(* Logix 5000 project; controller Amvex_Thorpe_Flowmeter vendor 1 type 14 code 106 rev 33.13; software revision 33.01; part 16 of 16 *)
(* tags used below, declared in another part *)
   Auto_Seq : SEQ;
   FAULTED : DINT;
   MODE : MODE;
   ID0_InputDataLength : MESSAGE;   // Message Command Input Data Data Length
   ID0_LengthParameterdata : MESSAGE;   // Message Command Parameter Data Length
   ID0_MSG_Diagnostic : MESSAGE;   // Message Get Diagnosis Module
   ID0_MSG_ProcessAlarm : MESSAGE;   // Message Get Get Process Alram Module
   ID0_OutputDataLength : MESSAGE;   // Message Command Output Data Data Length
   ID0_ReceiveMSG1 : MESSAGE;   // Message Command Parameter Receive Data
   ID0_ReceiveMSG2 : MESSAGE;   // Message Command Parameter Receive Data
   ID0_ReceiveMSG3 : MESSAGE;   // Message Command Parameter Receive Data
   ID0_SendMSG1 : MESSAGE;   // Message Command Parameter Send Data
   ID0_SendMSG2 : MESSAGE;   // Message Command Parameter Send Data
   ID0_SendMSG3 : MESSAGE;   // Message Command Parameter Send Data
   In_Cycle : BOOL;
   RCP1 : RCP1;
   RCP1_00 : UDT_ID0;
(* RPC1_Main, continued *)

ROUTINE R07_MODE   (* ladder *)
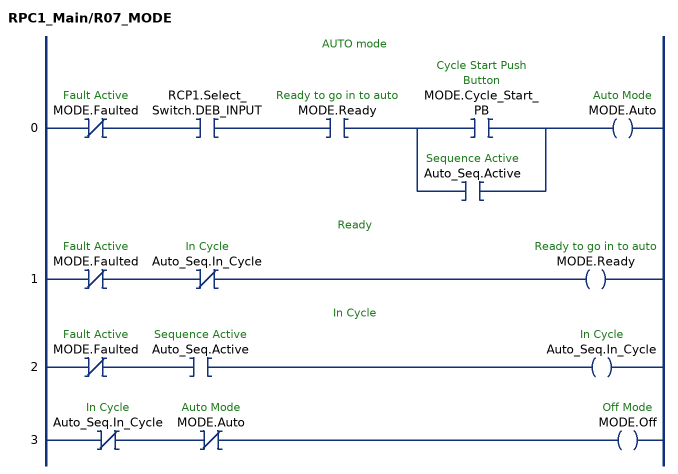
   // AUTO mode
   0: XIO(MODE.Faulted)XIC(RCP1.Select_Switch.DEB_INPUT)XIC(MODE.Ready)[XIC(MODE.Cycle_Start_PB) ,XIC(Auto_Seq.Active) ]OTE(MODE.Auto);
   // Ready
   1: XIO(MODE.Faulted)XIO(Auto_Seq.In_Cycle)OTE(MODE.Ready);
   // In Cycle
   2: XIO(MODE.Faulted)XIC(Auto_Seq.Active)OTE(Auto_Seq.In_Cycle);
   3: XIO(Auto_Seq.In_Cycle)XIO(MODE.Auto)OTE(MODE.Off);
END_ROUTINE

ROUTINE RCP1_00_RACK_IO   (* ladder *)
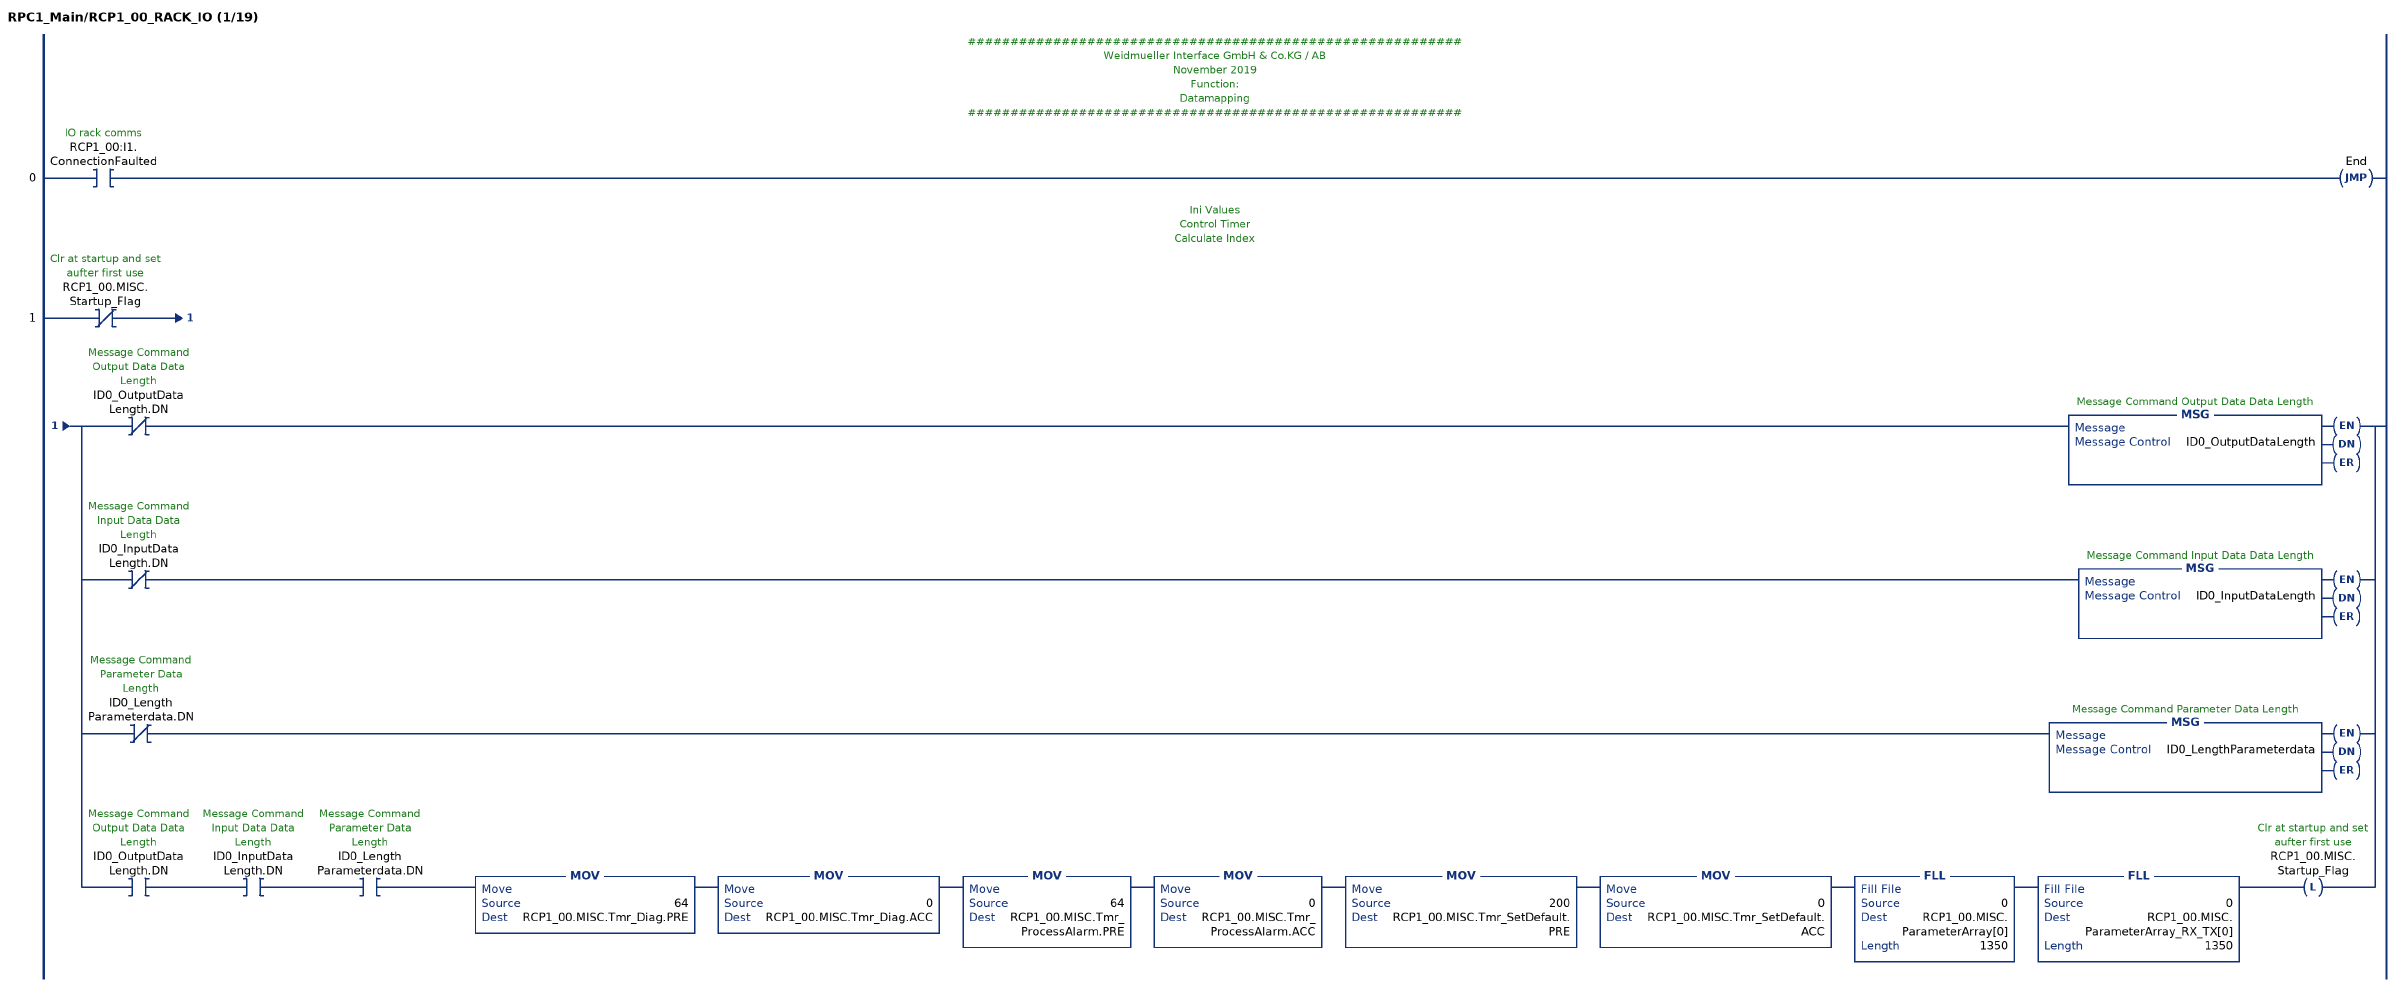
   // ##########################################################
   // Weidmueller Interface GmbH & Co.KG / AB
   // November 2019
   // Function:
   // Datamapping
   // ##########################################################
   0: XIC(RCP1_00:I1.ConnectionFaulted)JMP(End);
   // Ini Values
   // Control Timer
   // Calculate Index
   1: XIO(RCP1_00.MISC.Startup_Flag)[[XIO(ID0_OutputDataLength.DN) MSG(ID0_OutputDataLength) ,XIO(ID0_InputDataLength.DN) MSG(ID0_InputDataLength) ,XIO(ID0_LengthParameterdata.DN) MSG(ID0_LengthParameterdata) ] ,XIC(ID0_OutputDataLength.DN) XIC(ID0_InputDataLength.DN) XIC(ID0_LengthParameterdata.DN) MOV(64,RCP1_00.MISC.Tmr_Diag.PRE) MOV(0,RCP1_00.MISC.Tmr_Diag.ACC) MOV(64,RCP1_00.MISC.Tmr_ProcessAlarm.PRE) MOV(0,RCP1_00.MISC.Tmr_ProcessAlarm.ACC) MOV(200,RCP1_00.MISC.Tmr_SetDefault.PRE) MOV(0,RCP1_00.MISC.Tmr_SetDefault.ACC) FLL(0,RCP1_00.MISC.ParameterArray[0],1350) FLL(0,RCP1_00.MISC.ParameterArray_RX_TX[0],1350) OTL(RCP1_00.MISC.Startup_Flag) ];
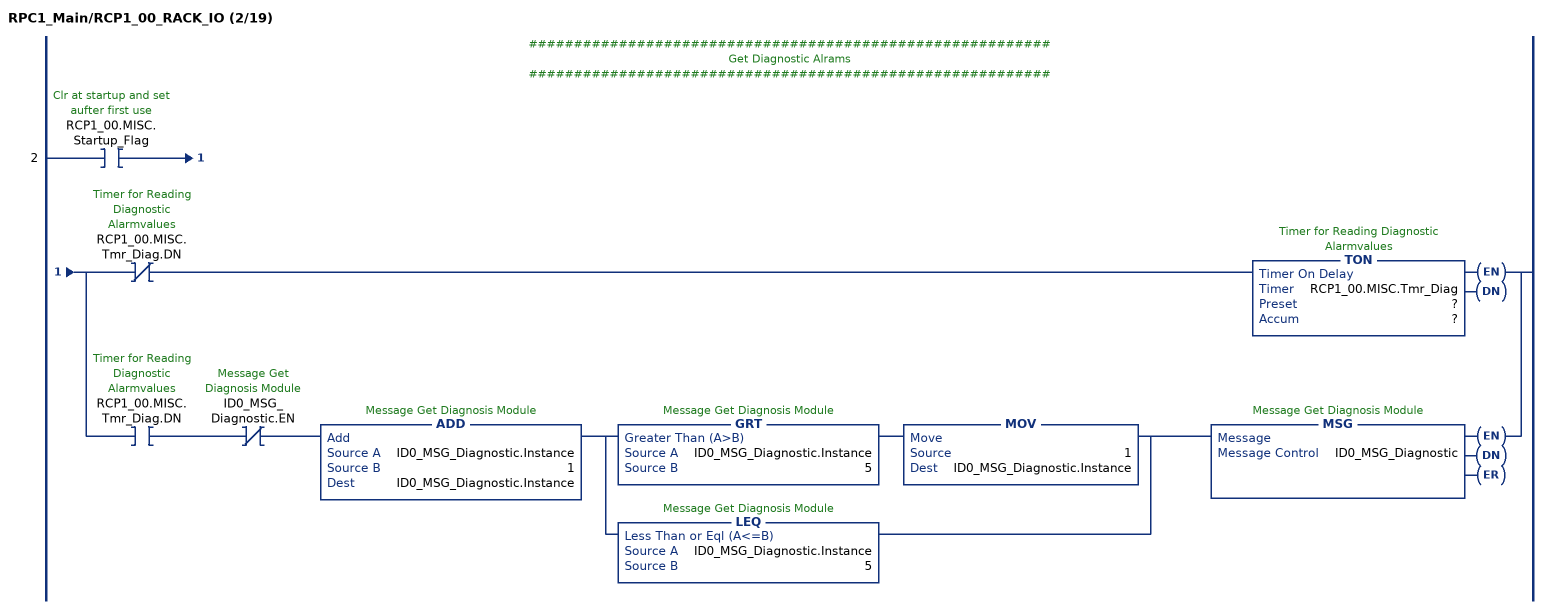
   // ##########################################################
   // Get Diagnostic Alrams
   // ##########################################################
   2: XIC(RCP1_00.MISC.Startup_Flag)[XIO(RCP1_00.MISC.Tmr_Diag.DN) TON(RCP1_00.MISC.Tmr_Diag,?,?) ,XIC(RCP1_00.MISC.Tmr_Diag.DN) XIO(ID0_MSG_Diagnostic.EN) ADD(ID0_MSG_Diagnostic.Instance,1,ID0_MSG_Diagnostic.Instance) [GRT(ID0_MSG_Diagnostic.Instance,5) MOV(1,ID0_MSG_Diagnostic.Instance) ,LEQ(ID0_MSG_Diagnostic.Instance,5) ] MSG(ID0_MSG_Diagnostic) ];
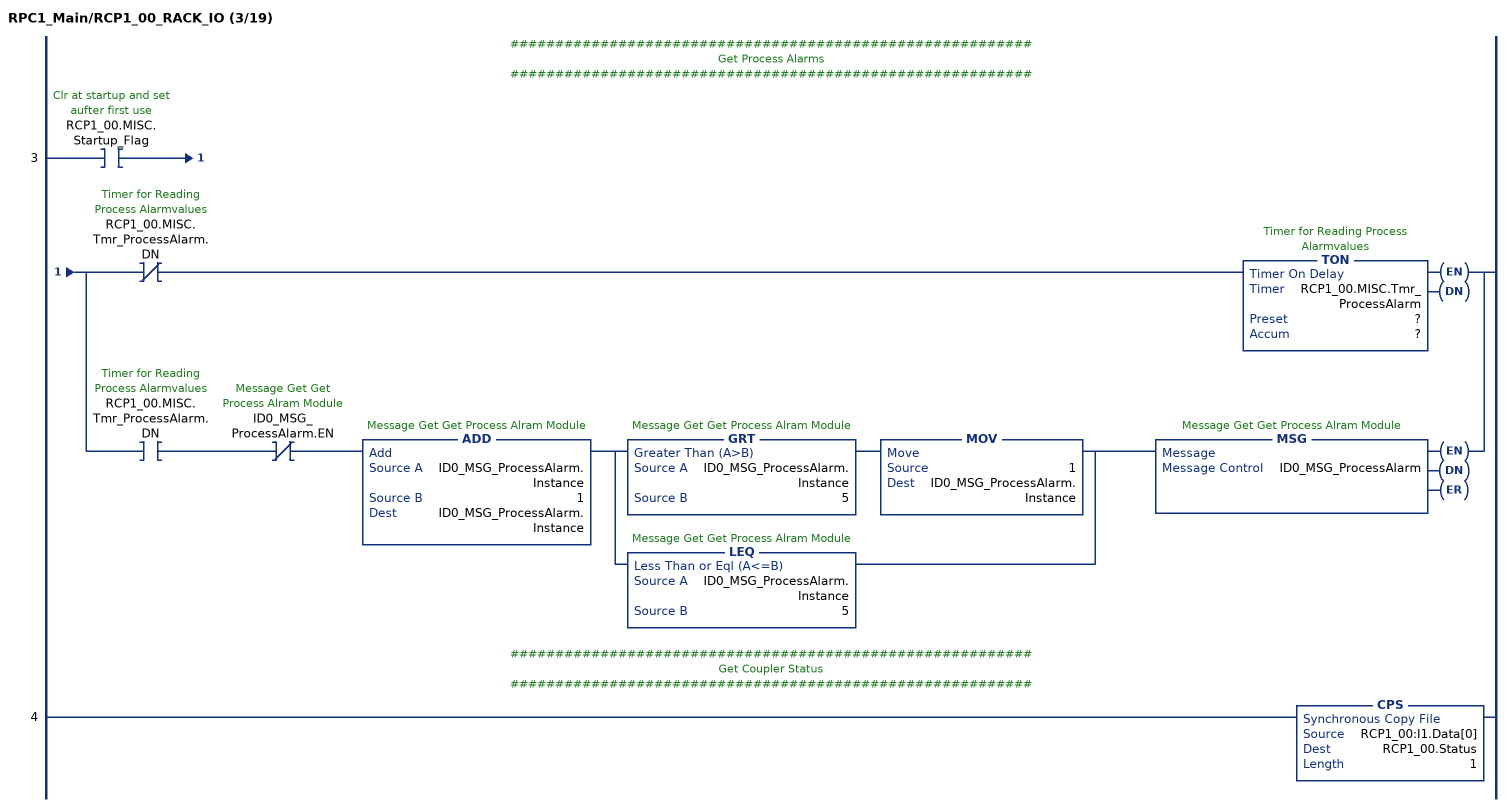
   // ##########################################################
   // Get Process Alarms
   // ##########################################################
   3: XIC(RCP1_00.MISC.Startup_Flag)[XIO(RCP1_00.MISC.Tmr_ProcessAlarm.DN) TON(RCP1_00.MISC.Tmr_ProcessAlarm,?,?) ,XIC(RCP1_00.MISC.Tmr_ProcessAlarm.DN) XIO(ID0_MSG_ProcessAlarm.EN) ADD(ID0_MSG_ProcessAlarm.Instance,1,ID0_MSG_ProcessAlarm.Instance) [GRT(ID0_MSG_ProcessAlarm.Instance,5) MOV(1,ID0_MSG_ProcessAlarm.Instance) ,LEQ(ID0_MSG_ProcessAlarm.Instance,5) ] MSG(ID0_MSG_ProcessAlarm) ];
   // ##########################################################
   // Get Coupler Status
   // ##########################################################
   4: CPS(RCP1_00:I1.Data[0],RCP1_00.Status,1);
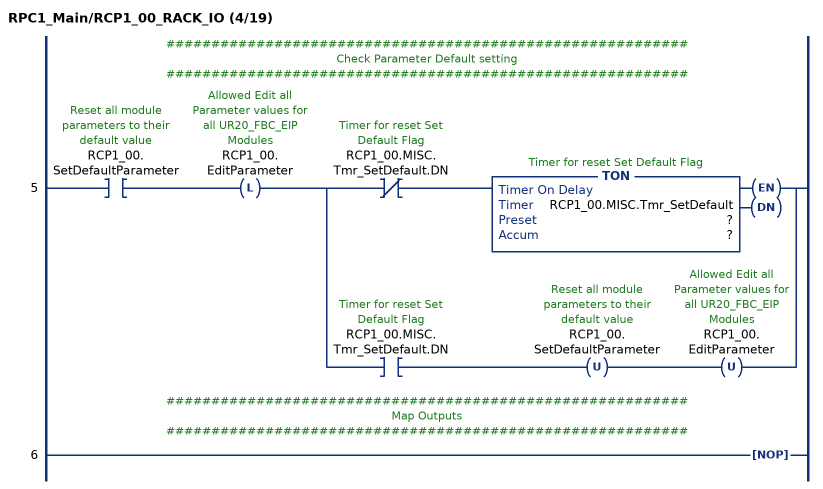
   // ##########################################################
   // Check Parameter Default setting
   // ##########################################################
   5: XIC(RCP1_00.SetDefaultParameter)OTL(RCP1_00.EditParameter)[XIO(RCP1_00.MISC.Tmr_SetDefault.DN) TON(RCP1_00.MISC.Tmr_SetDefault,?,?) ,XIC(RCP1_00.MISC.Tmr_SetDefault.DN) OTU(RCP1_00.SetDefaultParameter) OTU(RCP1_00.EditParameter) ];
   // ##########################################################
   // Map Outputs
   // ##########################################################
   6: NOP();
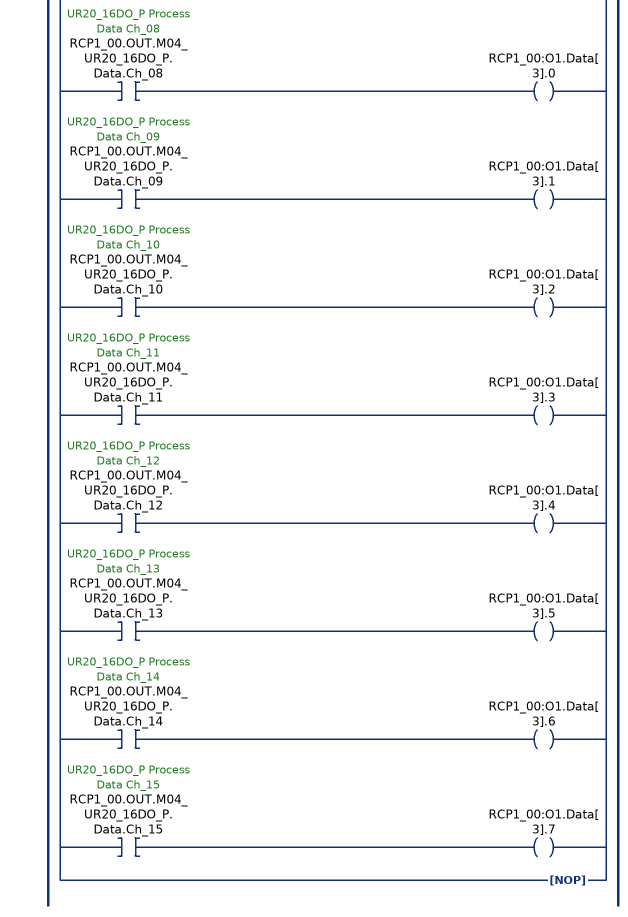
   // Map
   //  UR20_16DO_P
   //  Module No 4
   //  Process Data
   //  Outputs
   7: [NOP() ,XIC(RCP1_00.OUT.M04_UR20_16DO_P.Data.Ch_00) OTE(RCP1_00:O1.Data[2].0) ,XIC(RCP1_00.OUT.M04_UR20_16DO_P.Data.Ch_01) OTE(RCP1_00:O1.Data[2].1) ,XIC(RCP1_00.OUT.M04_UR20_16DO_P.Data.Ch_02) OTE(RCP1_00:O1.Data[2].2) ,XIC(RCP1_00.OUT.M04_UR20_16DO_P.Data.Ch_03) OTE(RCP1_00:O1.Data[2].3) ,XIC(RCP1_00.OUT.M04_UR20_16DO_P.Data.Ch_04) OTE(RCP1_00:O1.Data[2].4) ,XIC(RCP1_00.OUT.M04_UR20_16DO_P.Data.Ch_05) OTE(RCP1_00:O1.Data[2].5) ,XIC(RCP1_00.OUT.M04_UR20_16DO_P.Data.Ch_06) OTE(RCP1_00:O1.Data[2].6) ,XIC(RCP1_00.OUT.M04_UR20_16DO_P.Data.Ch_07) OTE(RCP1_00:O1.Data[2].7) ,XIC(RCP1_00.OUT.M04_UR20_16DO_P.Data.Ch_08) OTE(RCP1_00:O1.Data[3].0) ,XIC(RCP1_00.OUT.M04_UR20_16DO_P.Data.Ch_09) OTE(RCP1_00:O1.Data[3].1) ,XIC(RCP1_00.OUT.M04_UR20_16DO_P.Data.Ch_10) OTE(RCP1_00:O1.Data[3].2) ,XIC(RCP1_00.OUT.M04_UR20_16DO_P.Data.Ch_11) OTE(RCP1_00:O1.Data[3].3) ,XIC(RCP1_00.OUT.M04_UR20_16DO_P.Data.Ch_12) OTE(RCP1_00:O1.Data[3].4) ,XIC(RCP1_00.OUT.M04_UR20_16DO_P.Data.Ch_13) OTE(RCP1_00:O1.Data[3].5) ,XIC(RCP1_00.OUT.M04_UR20_16DO_P.Data.Ch_14) OTE(RCP1_00:O1.Data[3].6) ,XIC(RCP1_00.OUT.M04_UR20_16DO_P.Data.Ch_15) OTE(RCP1_00:O1.Data[3].7) ,NOP() ];
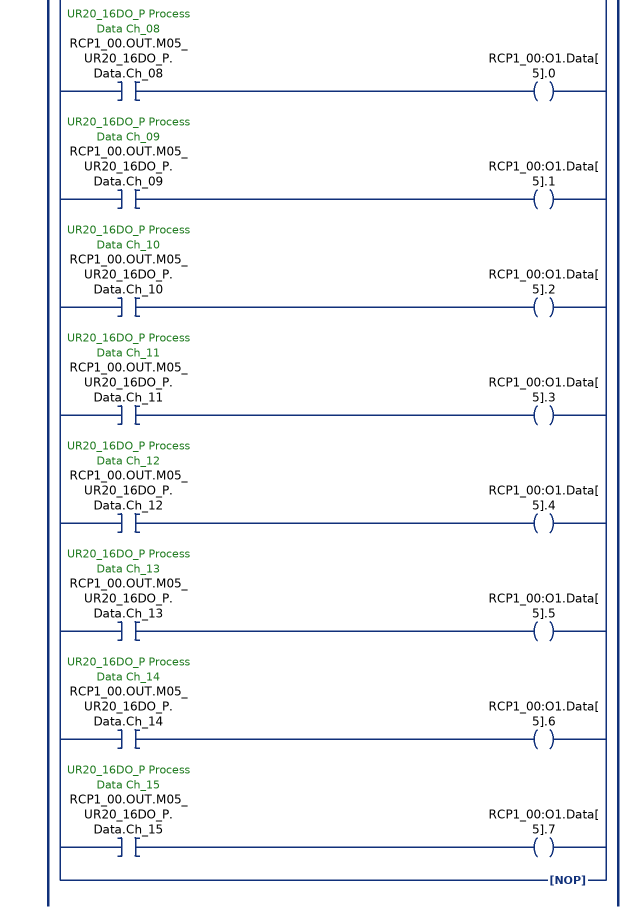
   // Map
   //  UR20_16DO_P
   //  Module No 5
   //  Process Data
   //  Outputs
   8: [NOP() ,XIC(RCP1_00.OUT.M05_UR20_16DO_P.Data.Ch_00) OTE(RCP1_00:O1.Data[4].0) ,XIC(RCP1_00.OUT.M05_UR20_16DO_P.Data.Ch_01) OTE(RCP1_00:O1.Data[4].1) ,XIC(RCP1_00.OUT.M05_UR20_16DO_P.Data.Ch_02) OTE(RCP1_00:O1.Data[4].2) ,XIC(RCP1_00.OUT.M05_UR20_16DO_P.Data.Ch_03) OTE(RCP1_00:O1.Data[4].3) ,XIC(RCP1_00.OUT.M05_UR20_16DO_P.Data.Ch_04) OTE(RCP1_00:O1.Data[4].4) ,XIC(RCP1_00.OUT.M05_UR20_16DO_P.Data.Ch_05) OTE(RCP1_00:O1.Data[4].5) ,XIC(RCP1_00.OUT.M05_UR20_16DO_P.Data.Ch_06) OTE(RCP1_00:O1.Data[4].6) ,XIC(RCP1_00.OUT.M05_UR20_16DO_P.Data.Ch_07) OTE(RCP1_00:O1.Data[4].7) ,XIC(RCP1_00.OUT.M05_UR20_16DO_P.Data.Ch_08) OTE(RCP1_00:O1.Data[5].0) ,XIC(RCP1_00.OUT.M05_UR20_16DO_P.Data.Ch_09) OTE(RCP1_00:O1.Data[5].1) ,XIC(RCP1_00.OUT.M05_UR20_16DO_P.Data.Ch_10) OTE(RCP1_00:O1.Data[5].2) ,XIC(RCP1_00.OUT.M05_UR20_16DO_P.Data.Ch_11) OTE(RCP1_00:O1.Data[5].3) ,XIC(RCP1_00.OUT.M05_UR20_16DO_P.Data.Ch_12) OTE(RCP1_00:O1.Data[5].4) ,XIC(RCP1_00.OUT.M05_UR20_16DO_P.Data.Ch_13) OTE(RCP1_00:O1.Data[5].5) ,XIC(RCP1_00.OUT.M05_UR20_16DO_P.Data.Ch_14) OTE(RCP1_00:O1.Data[5].6) ,XIC(RCP1_00.OUT.M05_UR20_16DO_P.Data.Ch_15) OTE(RCP1_00:O1.Data[5].7) ,NOP() ];
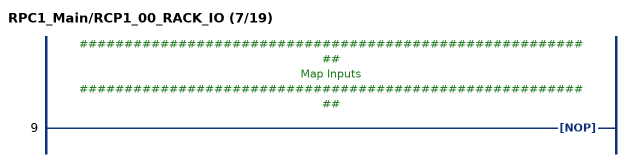
   // ##########################################################
   // Map Inputs
   // ##########################################################
   9: NOP();
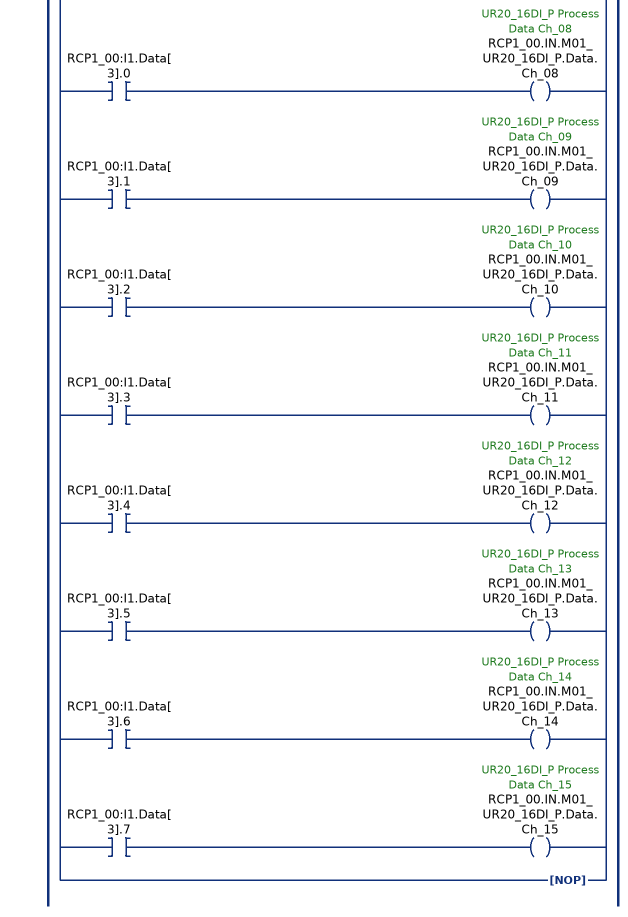
   // Map
   //  UR20_16DI_P
   //  Module No 1
   //  Process Data
   //  Inputs
   10: [NOP() ,XIC(RCP1_00:I1.Data[2].0) OTE(RCP1_00.IN.M01_UR20_16DI_P.Data.Ch_00) ,XIC(RCP1_00:I1.Data[2].1) OTE(RCP1_00.IN.M01_UR20_16DI_P.Data.Ch_01) ,XIC(RCP1_00:I1.Data[2].2) OTE(RCP1_00.IN.M01_UR20_16DI_P.Data.Ch_02) ,XIC(RCP1_00:I1.Data[2].3) OTE(RCP1_00.IN.M01_UR20_16DI_P.Data.Ch_03) ,XIC(RCP1_00:I1.Data[2].4) OTE(RCP1_00.IN.M01_UR20_16DI_P.Data.Ch_04) ,XIC(RCP1_00:I1.Data[2].5) OTE(RCP1_00.IN.M01_UR20_16DI_P.Data.Ch_05) ,XIC(RCP1_00:I1.Data[2].6) OTE(RCP1_00.IN.M01_UR20_16DI_P.Data.Ch_06) ,XIC(RCP1_00:I1.Data[2].7) OTE(RCP1_00.IN.M01_UR20_16DI_P.Data.Ch_07) ,XIC(RCP1_00:I1.Data[3].0) OTE(RCP1_00.IN.M01_UR20_16DI_P.Data.Ch_08) ,XIC(RCP1_00:I1.Data[3].1) OTE(RCP1_00.IN.M01_UR20_16DI_P.Data.Ch_09) ,XIC(RCP1_00:I1.Data[3].2) OTE(RCP1_00.IN.M01_UR20_16DI_P.Data.Ch_10) ,XIC(RCP1_00:I1.Data[3].3) OTE(RCP1_00.IN.M01_UR20_16DI_P.Data.Ch_11) ,XIC(RCP1_00:I1.Data[3].4) OTE(RCP1_00.IN.M01_UR20_16DI_P.Data.Ch_12) ,XIC(RCP1_00:I1.Data[3].5) OTE(RCP1_00.IN.M01_UR20_16DI_P.Data.Ch_13) ,XIC(RCP1_00:I1.Data[3].6) OTE(RCP1_00.IN.M01_UR20_16DI_P.Data.Ch_14) ,XIC(RCP1_00:I1.Data[3].7) OTE(RCP1_00.IN.M01_UR20_16DI_P.Data.Ch_15) ,NOP() ];
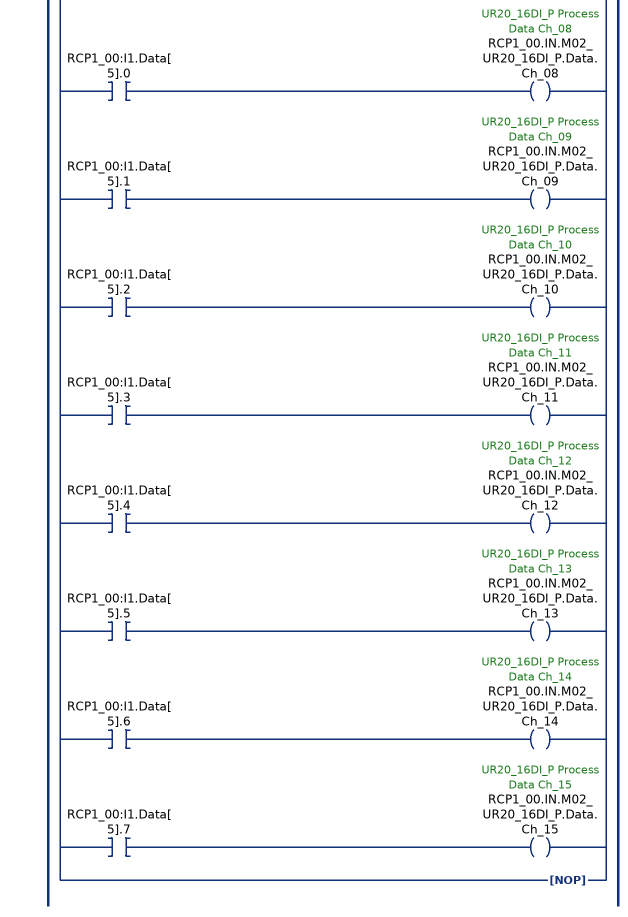
   // Map
   //  UR20_16DI_P
   //  Module No 2
   //  Process Data
   //  Inputs
   11: [NOP() ,XIC(RCP1_00:I1.Data[4].0) OTE(RCP1_00.IN.M02_UR20_16DI_P.Data.Ch_00) ,XIC(RCP1_00:I1.Data[4].1) OTE(RCP1_00.IN.M02_UR20_16DI_P.Data.Ch_01) ,XIC(RCP1_00:I1.Data[4].2) OTE(RCP1_00.IN.M02_UR20_16DI_P.Data.Ch_02) ,XIC(RCP1_00:I1.Data[4].3) OTE(RCP1_00.IN.M02_UR20_16DI_P.Data.Ch_03) ,XIC(RCP1_00:I1.Data[4].4) OTE(RCP1_00.IN.M02_UR20_16DI_P.Data.Ch_04) ,XIC(RCP1_00:I1.Data[4].5) OTE(RCP1_00.IN.M02_UR20_16DI_P.Data.Ch_05) ,XIC(RCP1_00:I1.Data[4].6) OTE(RCP1_00.IN.M02_UR20_16DI_P.Data.Ch_06) ,XIC(RCP1_00:I1.Data[4].7) OTE(RCP1_00.IN.M02_UR20_16DI_P.Data.Ch_07) ,XIC(RCP1_00:I1.Data[5].0) OTE(RCP1_00.IN.M02_UR20_16DI_P.Data.Ch_08) ,XIC(RCP1_00:I1.Data[5].1) OTE(RCP1_00.IN.M02_UR20_16DI_P.Data.Ch_09) ,XIC(RCP1_00:I1.Data[5].2) OTE(RCP1_00.IN.M02_UR20_16DI_P.Data.Ch_10) ,XIC(RCP1_00:I1.Data[5].3) OTE(RCP1_00.IN.M02_UR20_16DI_P.Data.Ch_11) ,XIC(RCP1_00:I1.Data[5].4) OTE(RCP1_00.IN.M02_UR20_16DI_P.Data.Ch_12) ,XIC(RCP1_00:I1.Data[5].5) OTE(RCP1_00.IN.M02_UR20_16DI_P.Data.Ch_13) ,XIC(RCP1_00:I1.Data[5].6) OTE(RCP1_00.IN.M02_UR20_16DI_P.Data.Ch_14) ,XIC(RCP1_00:I1.Data[5].7) OTE(RCP1_00.IN.M02_UR20_16DI_P.Data.Ch_15) ,NOP() ];
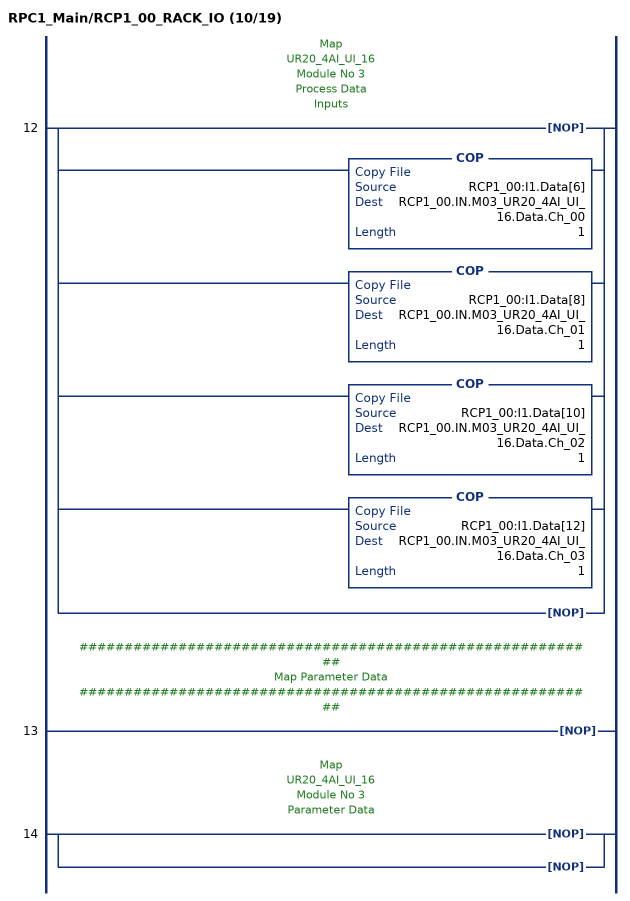
   // Map
   //  UR20_4AI_UI_16
   //  Module No 3
   //  Process Data
   //  Inputs
   12: [NOP() ,COP(RCP1_00:I1.Data[6],RCP1_00.IN.M03_UR20_4AI_UI_16.Data.Ch_00,1) ,COP(RCP1_00:I1.Data[8],RCP1_00.IN.M03_UR20_4AI_UI_16.Data.Ch_01,1) ,COP(RCP1_00:I1.Data[10],RCP1_00.IN.M03_UR20_4AI_UI_16.Data.Ch_02,1) ,COP(RCP1_00:I1.Data[12],RCP1_00.IN.M03_UR20_4AI_UI_16.Data.Ch_03,1) ,NOP() ];
   // ##########################################################
   // Map Parameter Data
   // ##########################################################
   13: NOP();
   // Map
   //  UR20_4AI_UI_16
   //  Module No 3
   //  Parameter Data
   14: [NOP() ,NOP() ];
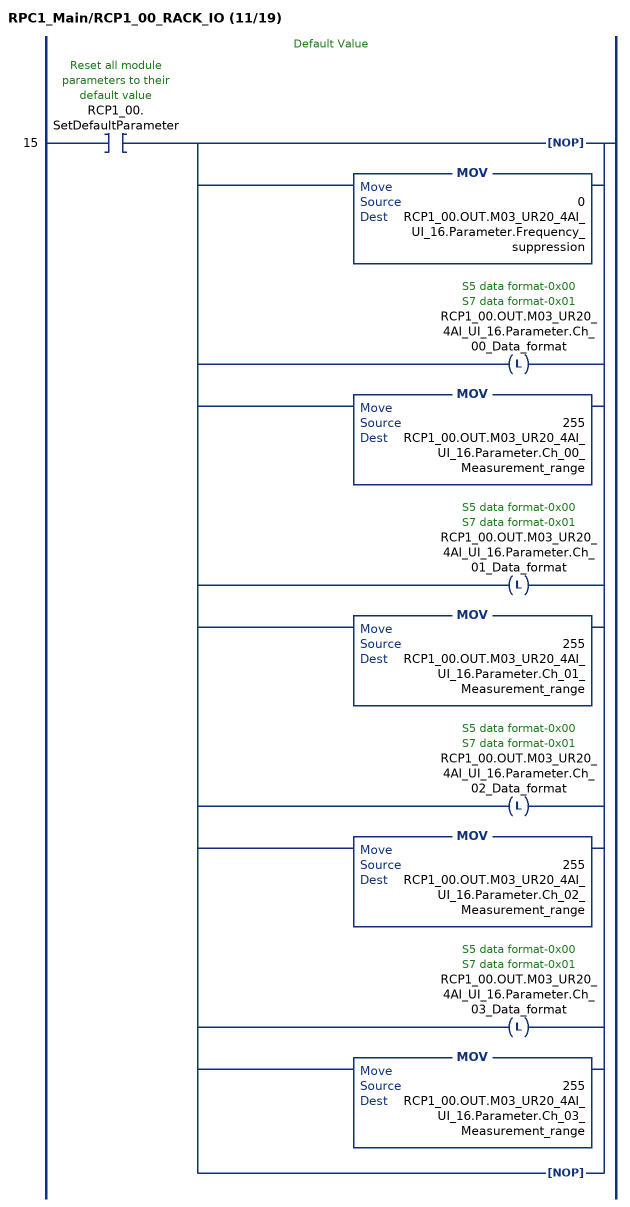
   // Default Value
   15: XIC(RCP1_00.SetDefaultParameter)[NOP() ,MOV(0,RCP1_00.OUT.M03_UR20_4AI_UI_16.Parameter.Frequency_suppression) ,OTL(RCP1_00.OUT.M03_UR20_4AI_UI_16.Parameter.Ch_00_Data_format) ,MOV(255,RCP1_00.OUT.M03_UR20_4AI_UI_16.Parameter.Ch_00_Measurement_range) ,OTL(RCP1_00.OUT.M03_UR20_4AI_UI_16.Parameter.Ch_01_Data_format) ,MOV(255,RCP1_00.OUT.M03_UR20_4AI_UI_16.Parameter.Ch_01_Measurement_range) ,OTL(RCP1_00.OUT.M03_UR20_4AI_UI_16.Parameter.Ch_02_Data_format) ,MOV(255,RCP1_00.OUT.M03_UR20_4AI_UI_16.Parameter.Ch_02_Measurement_range) ,OTL(RCP1_00.OUT.M03_UR20_4AI_UI_16.Parameter.Ch_03_Data_format) ,MOV(255,RCP1_00.OUT.M03_UR20_4AI_UI_16.Parameter.Ch_03_Measurement_range) ,NOP() ];
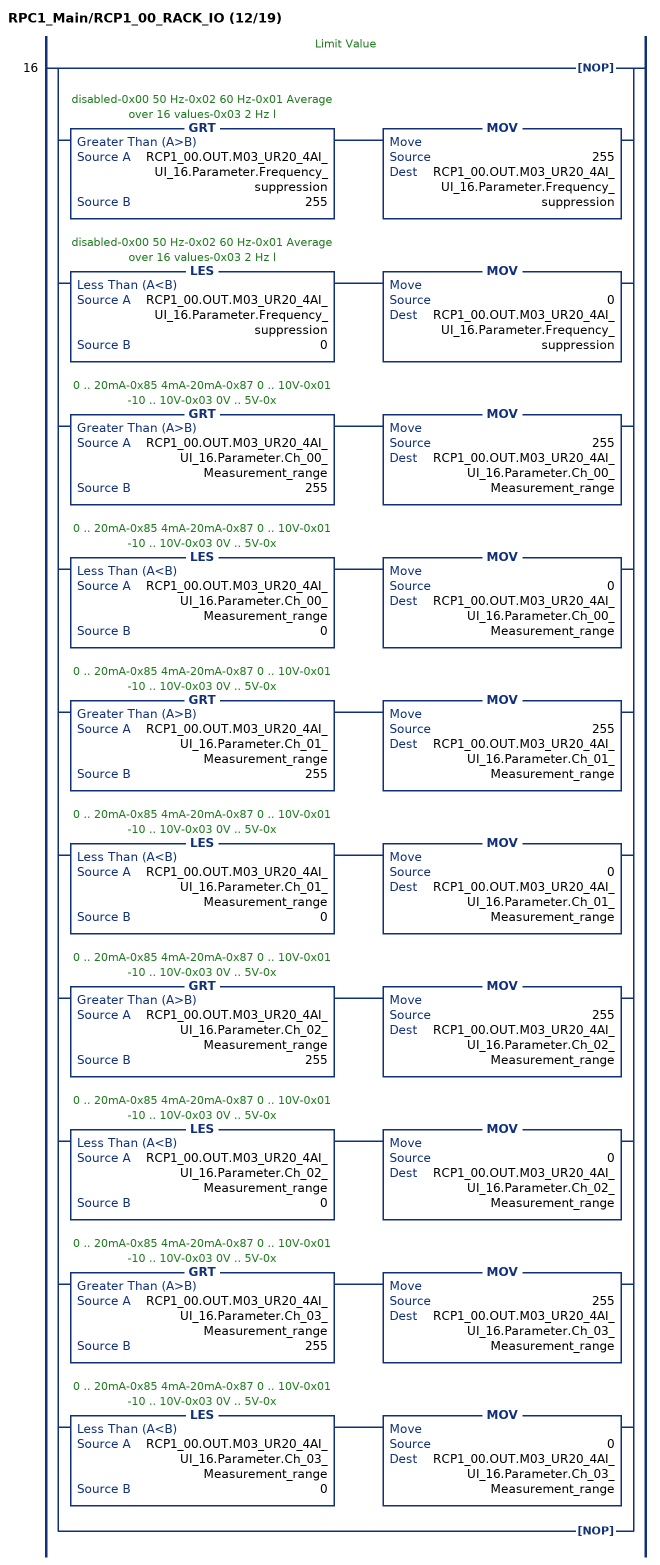
   // Limit Value
   16: [NOP() ,GRT(RCP1_00.OUT.M03_UR20_4AI_UI_16.Parameter.Frequency_suppression,255) MOV(255,RCP1_00.OUT.M03_UR20_4AI_UI_16.Parameter.Frequency_suppression) ,LES(RCP1_00.OUT.M03_UR20_4AI_UI_16.Parameter.Frequency_suppression,0) MOV(0,RCP1_00.OUT.M03_UR20_4AI_UI_16.Parameter.Frequency_suppression) ,GRT(RCP1_00.OUT.M03_UR20_4AI_UI_16.Parameter.Ch_00_Measurement_range,255) MOV(255,RCP1_00.OUT.M03_UR20_4AI_UI_16.Parameter.Ch_00_Measurement_range) ,LES(RCP1_00.OUT.M03_UR20_4AI_UI_16.Parameter.Ch_00_Measurement_range,0) MOV(0,RCP1_00.OUT.M03_UR20_4AI_UI_16.Parameter.Ch_00_Measurement_range) ,GRT(RCP1_00.OUT.M03_UR20_4AI_UI_16.Parameter.Ch_01_Measurement_range,255) MOV(255,RCP1_00.OUT.M03_UR20_4AI_UI_16.Parameter.Ch_01_Measurement_range) ,LES(RCP1_00.OUT.M03_UR20_4AI_UI_16.Parameter.Ch_01_Measurement_range,0) MOV(0,RCP1_00.OUT.M03_UR20_4AI_UI_16.Parameter.Ch_01_Measurement_range) ,GRT(RCP1_00.OUT.M03_UR20_4AI_UI_16.Parameter.Ch_02_Measurement_range,255) MOV(255,RCP1_00.OUT.M03_UR20_4AI_UI_16.Parameter.Ch_02_Measurement_range) ,LES(RCP1_00.OUT.M03_UR20_4AI_UI_16.Parameter.Ch_02_Measurement_range,0) MOV(0,RCP1_00.OUT.M03_UR20_4AI_UI_16.Parameter.Ch_02_Measurement_range) ,GRT(RCP1_00.OUT.M03_UR20_4AI_UI_16.Parameter.Ch_03_Measurement_range,255) MOV(255,RCP1_00.OUT.M03_UR20_4AI_UI_16.Parameter.Ch_03_Measurement_range) ,LES(RCP1_00.OUT.M03_UR20_4AI_UI_16.Parameter.Ch_03_Measurement_range,0) MOV(0,RCP1_00.OUT.M03_UR20_4AI_UI_16.Parameter.Ch_03_Measurement_range) ,NOP() ];
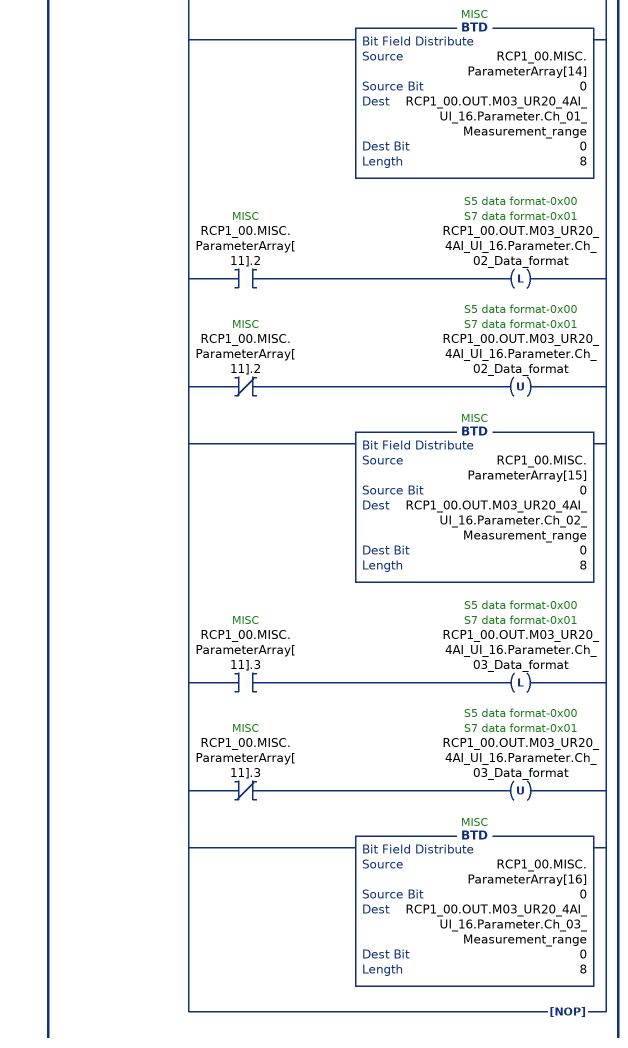
   // Read Parameter from Module
   17: XIO(RCP1_00.EditParameter)[NOP() ,BTD(RCP1_00.MISC.ParameterArray[12],0,RCP1_00.OUT.M03_UR20_4AI_UI_16.Parameter.Frequency_suppression,0,8) ,XIC(RCP1_00.MISC.ParameterArray[11].0) OTL(RCP1_00.OUT.M03_UR20_4AI_UI_16.Parameter.Ch_00_Data_format) ,XIO(RCP1_00.MISC.ParameterArray[11].0) OTU(RCP1_00.OUT.M03_UR20_4AI_UI_16.Parameter.Ch_00_Data_format) ,BTD(RCP1_00.MISC.ParameterArray[13],0,RCP1_00.OUT.M03_UR20_4AI_UI_16.Parameter.Ch_00_Measurement_range,0,8) ,XIC(RCP1_00.MISC.ParameterArray[11].1) OTL(RCP1_00.OUT.M03_UR20_4AI_UI_16.Parameter.Ch_01_Data_format) ,XIO(RCP1_00.MISC.ParameterArray[11].1) OTU(RCP1_00.OUT.M03_UR20_4AI_UI_16.Parameter.Ch_01_Data_format) ,BTD(RCP1_00.MISC.ParameterArray[14],0,RCP1_00.OUT.M03_UR20_4AI_UI_16.Parameter.Ch_01_Measurement_range,0,8) ,XIC(RCP1_00.MISC.ParameterArray[11].2) OTL(RCP1_00.OUT.M03_UR20_4AI_UI_16.Parameter.Ch_02_Data_format) ,XIO(RCP1_00.MISC.ParameterArray[11].2) OTU(RCP1_00.OUT.M03_UR20_4AI_UI_16.Parameter.Ch_02_Data_format) ,BTD(RCP1_00.MISC.ParameterArray[15],0,RCP1_00.OUT.M03_UR20_4AI_UI_16.Parameter.Ch_02_Measurement_range,0,8) ,XIC(RCP1_00.MISC.ParameterArray[11].3) OTL(RCP1_00.OUT.M03_UR20_4AI_UI_16.Parameter.Ch_03_Data_format) ,XIO(RCP1_00.MISC.ParameterArray[11].3) OTU(RCP1_00.OUT.M03_UR20_4AI_UI_16.Parameter.Ch_03_Data_format) ,BTD(RCP1_00.MISC.ParameterArray[16],0,RCP1_00.OUT.M03_UR20_4AI_UI_16.Parameter.Ch_03_Measurement_range,0,8) ,NOP() ];
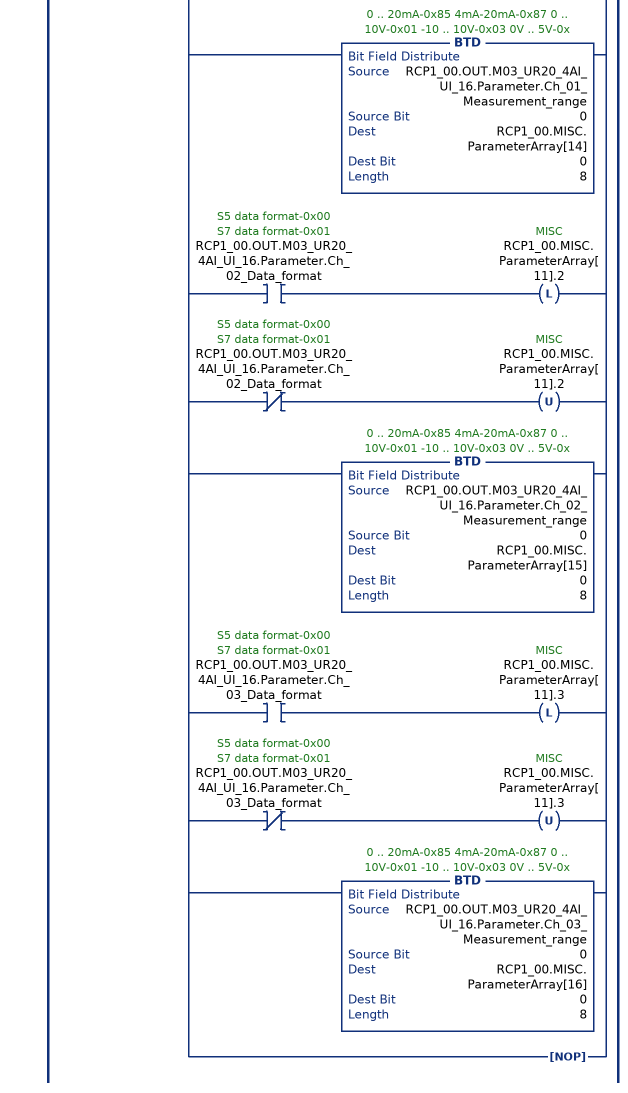
   // Write Parameter to Module
   18: XIC(RCP1_00.EditParameter)[NOP() ,BTD(RCP1_00.OUT.M03_UR20_4AI_UI_16.Parameter.Frequency_suppression,0,RCP1_00.MISC.ParameterArray[12],0,8) ,XIC(RCP1_00.OUT.M03_UR20_4AI_UI_16.Parameter.Ch_00_Data_format) OTL(RCP1_00.MISC.ParameterArray[11].0) ,XIO(RCP1_00.OUT.M03_UR20_4AI_UI_16.Parameter.Ch_00_Data_format) OTU(RCP1_00.MISC.ParameterArray[11].0) ,BTD(RCP1_00.OUT.M03_UR20_4AI_UI_16.Parameter.Ch_00_Measurement_range,0,RCP1_00.MISC.ParameterArray[13],0,8) ,XIC(RCP1_00.OUT.M03_UR20_4AI_UI_16.Parameter.Ch_01_Data_format) OTL(RCP1_00.MISC.ParameterArray[11].1) ,XIO(RCP1_00.OUT.M03_UR20_4AI_UI_16.Parameter.Ch_01_Data_format) OTU(RCP1_00.MISC.ParameterArray[11].1) ,BTD(RCP1_00.OUT.M03_UR20_4AI_UI_16.Parameter.Ch_01_Measurement_range,0,RCP1_00.MISC.ParameterArray[14],0,8) ,XIC(RCP1_00.OUT.M03_UR20_4AI_UI_16.Parameter.Ch_02_Data_format) OTL(RCP1_00.MISC.ParameterArray[11].2) ,XIO(RCP1_00.OUT.M03_UR20_4AI_UI_16.Parameter.Ch_02_Data_format) OTU(RCP1_00.MISC.ParameterArray[11].2) ,BTD(RCP1_00.OUT.M03_UR20_4AI_UI_16.Parameter.Ch_02_Measurement_range,0,RCP1_00.MISC.ParameterArray[15],0,8) ,XIC(RCP1_00.OUT.M03_UR20_4AI_UI_16.Parameter.Ch_03_Data_format) OTL(RCP1_00.MISC.ParameterArray[11].3) ,XIO(RCP1_00.OUT.M03_UR20_4AI_UI_16.Parameter.Ch_03_Data_format) OTU(RCP1_00.MISC.ParameterArray[11].3) ,BTD(RCP1_00.OUT.M03_UR20_4AI_UI_16.Parameter.Ch_03_Measurement_range,0,RCP1_00.MISC.ParameterArray[16],0,8) ,NOP() ];
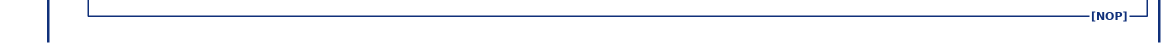
   // ##########################################################
   // DiagnoseAlarm Daten
   // ##########################################################
   19: XIC(ID0_MSG_Diagnostic.DN)[NOP() ,EQU(ID0_MSG_Diagnostic.Instance,1) [NEQ(RCP1_00.MISC.DiagnosticData[0],0) OTL(RCP1_00.IN.M01_UR20_16DI_P.StatusDiagAlarm) ,EQU(RCP1_00.MISC.DiagnosticData[0],0) OTU(RCP1_00.IN.M01_UR20_16DI_P.StatusDiagAlarm) ] CPS(RCP1_00.MISC.DiagnosticData[0],RCP1_00.IN.M01_UR20_16DI_P.Diagnostic,1) ,EQU(ID0_MSG_Diagnostic.Instance,2) [NEQ(RCP1_00.MISC.DiagnosticData[0],0) OTL(RCP1_00.IN.M02_UR20_16DI_P.StatusDiagAlarm) ,EQU(RCP1_00.MISC.DiagnosticData[0],0) OTU(RCP1_00.IN.M02_UR20_16DI_P.StatusDiagAlarm) ] CPS(RCP1_00.MISC.DiagnosticData[0],RCP1_00.IN.M02_UR20_16DI_P.Diagnostic,1) ,EQU(ID0_MSG_Diagnostic.Instance,3) [NEQ(RCP1_00.MISC.DiagnosticData[0],0) OTL(RCP1_00.IN.M03_UR20_4AI_UI_16.StatusDiagAlarm) ,EQU(RCP1_00.MISC.DiagnosticData[0],0) OTU(RCP1_00.IN.M03_UR20_4AI_UI_16.StatusDiagAlarm) ] CPS(RCP1_00.MISC.DiagnosticData[0],RCP1_00.IN.M03_UR20_4AI_UI_16.Diagnostic,1) ,EQU(ID0_MSG_Diagnostic.Instance,4) [NEQ(RCP1_00.MISC.DiagnosticData[0],0) OTL(RCP1_00.IN.M04_UR20_16DO_P.StatusDiagAlarm) ,EQU(RCP1_00.MISC.DiagnosticData[0],0) OTU(RCP1_00.IN.M04_UR20_16DO_P.StatusDiagAlarm) ] CPS(RCP1_00.MISC.DiagnosticData[0],RCP1_00.IN.M04_UR20_16DO_P.Diagnostic,1) ,EQU(ID0_MSG_Diagnostic.Instance,5) [NEQ(RCP1_00.MISC.DiagnosticData[0],0) OTL(RCP1_00.IN.M05_UR20_16DO_P.StatusDiagAlarm) ,EQU(RCP1_00.MISC.DiagnosticData[0],0) OTU(RCP1_00.IN.M05_UR20_16DO_P.StatusDiagAlarm) ] CPS(RCP1_00.MISC.DiagnosticData[0],RCP1_00.IN.M05_UR20_16DO_P.Diagnostic,1) ,NOP() ];
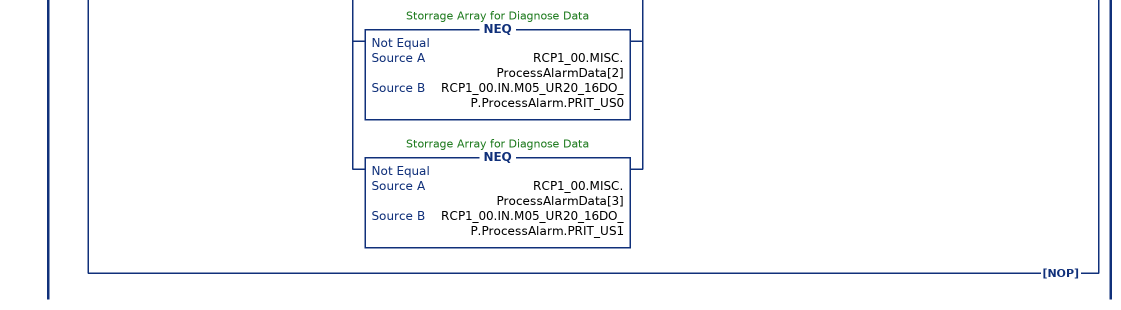
   // ##########################################################
   // ProcessAlarm Daten
   // ##########################################################
   20: XIC(ID0_MSG_ProcessAlarm.DN)[NOP() ,EQU(ID0_MSG_ProcessAlarm.Instance,1) [NEQ(RCP1_00.MISC.ProcessAlarmData[0],RCP1_00.IN.M01_UR20_16DI_P.ProcessAlarm.PRIT_OL) ,NEQ(RCP1_00.MISC.ProcessAlarmData[1],RCP1_00.IN.M01_UR20_16DI_P.ProcessAlarm.PRIT_UL) ,NEQ(RCP1_00.MISC.ProcessAlarmData[2],RCP1_00.IN.M01_UR20_16DI_P.ProcessAlarm.PRIT_US0) ,NEQ(RCP1_00.MISC.ProcessAlarmData[3],RCP1_00.IN.M01_UR20_16DI_P.ProcessAlarm.PRIT_US1) ] OTL(RCP1_00.IN.M01_UR20_16DI_P.StatusProcessAlarm) CPS(RCP1_00.MISC.ProcessAlarmData[0],RCP1_00.IN.M01_UR20_16DI_P.ProcessAlarm,1) ,EQU(ID0_MSG_ProcessAlarm.Instance,2) [NEQ(RCP1_00.MISC.ProcessAlarmData[0],RCP1_00.IN.M02_UR20_16DI_P.ProcessAlarm.PRIT_OL) ,NEQ(RCP1_00.MISC.ProcessAlarmData[1],RCP1_00.IN.M02_UR20_16DI_P.ProcessAlarm.PRIT_UL) ,NEQ(RCP1_00.MISC.ProcessAlarmData[2],RCP1_00.IN.M02_UR20_16DI_P.ProcessAlarm.PRIT_US0) ,NEQ(RCP1_00.MISC.ProcessAlarmData[3],RCP1_00.IN.M02_UR20_16DI_P.ProcessAlarm.PRIT_US1) ] OTL(RCP1_00.IN.M02_UR20_16DI_P.StatusProcessAlarm) CPS(RCP1_00.MISC.ProcessAlarmData[0],RCP1_00.IN.M02_UR20_16DI_P.ProcessAlarm,1) ,EQU(ID0_MSG_ProcessAlarm.Instance,3) [NEQ(RCP1_00.MISC.ProcessAlarmData[0],RCP1_00.IN.M03_UR20_4AI_UI_16.ProcessAlarm.PRIT_OL) ,NEQ(RCP1_00.MISC.ProcessAlarmData[1],RCP1_00.IN.M03_UR20_4AI_UI_16.ProcessAlarm.PRIT_UL) ,NEQ(RCP1_00.MISC.ProcessAlarmData[2],RCP1_00.IN.M03_UR20_4AI_UI_16.ProcessAlarm.PRIT_US0) ,NEQ(RCP1_00.MISC.ProcessAlarmData[3],RCP1_00.IN.M03_UR20_4AI_UI_16.ProcessAlarm.PRIT_US1) ] OTL(RCP1_00.IN.M03_UR20_4AI_UI_16.StatusProcessAlarm) CPS(RCP1_00.MISC.ProcessAlarmData[0],RCP1_00.IN.M03_UR20_4AI_UI_16.ProcessAlarm,1) ,EQU(ID0_MSG_ProcessAlarm.Instance,4) [NEQ(RCP1_00.MISC.ProcessAlarmData[0],RCP1_00.IN.M04_UR20_16DO_P.ProcessAlarm.PRIT_OL) ,NEQ(RCP1_00.MISC.ProcessAlarmData[1],RCP1_00.IN.M04_UR20_16DO_P.ProcessAlarm.PRIT_UL) ,NEQ(RCP1_00.MISC.ProcessAlarmData[2],RCP1_00.IN.M04_UR20_16DO_P.ProcessAlarm.PRIT_US0) ,NEQ(RCP1_00.MISC.ProcessAlarmData[3],RCP1_00.IN.M04_UR20_16DO_P.ProcessAlarm.PRIT_US1) ] OTL(RCP1_00.IN.M04_UR20_16DO_P.StatusProcessAlarm) CPS(RCP1_00.MISC.ProcessAlarmData[0],RCP1_00.IN.M04_UR20_16DO_P.ProcessAlarm,1) ,EQU(ID0_MSG_ProcessAlarm.Instance,5) [NEQ(RCP1_00.MISC.ProcessAlarmData[0],RCP1_00.IN.M05_UR20_16DO_P.ProcessAlarm.PRIT_OL) ,NEQ(RCP1_00.MISC.ProcessAlarmData[1],RCP1_00.IN.M05_UR20_16DO_P.ProcessAlarm.PRIT_UL) ,NEQ(RCP1_00.MISC.ProcessAlarmData[2],RCP1_00.IN.M05_UR20_16DO_P.ProcessAlarm.PRIT_US0) ,NEQ(RCP1_00.MISC.ProcessAlarmData[3],RCP1_00.IN.M05_UR20_16DO_P.ProcessAlarm.PRIT_US1) ] OTL(RCP1_00.IN.M05_UR20_16DO_P.StatusProcessAlarm) CPS(RCP1_00.MISC.ProcessAlarmData[0],RCP1_00.IN.M05_UR20_16DO_P.ProcessAlarm,1) ,NOP() ];
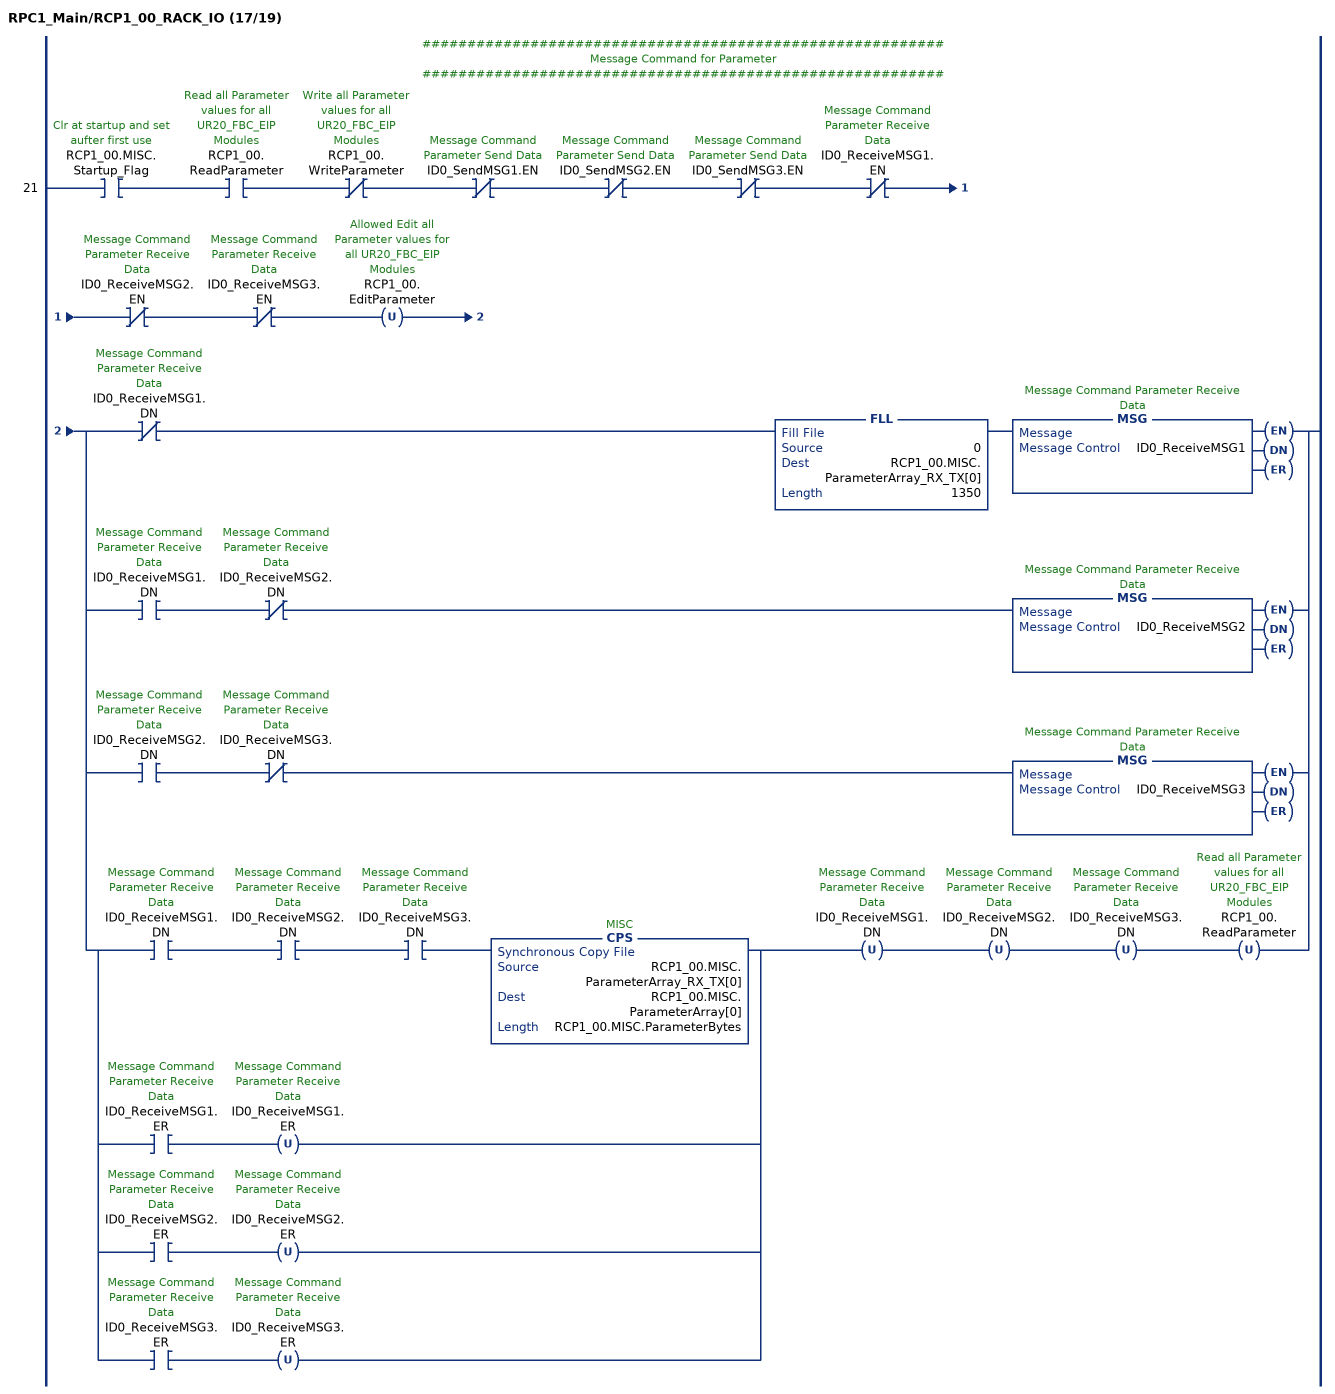
   // ##########################################################
   // Message Command for Parameter
   // ##########################################################
   21: XIC(RCP1_00.MISC.Startup_Flag)XIC(RCP1_00.ReadParameter)XIO(RCP1_00.WriteParameter)XIO(ID0_SendMSG1.EN)XIO(ID0_SendMSG2.EN)XIO(ID0_SendMSG3.EN)XIO(ID0_ReceiveMSG1.EN)XIO(ID0_ReceiveMSG2.EN)XIO(ID0_ReceiveMSG3.EN)OTU(RCP1_00.EditParameter)[XIO(ID0_ReceiveMSG1.DN) FLL(0,RCP1_00.MISC.ParameterArray_RX_TX[0],1350) MSG(ID0_ReceiveMSG1) ,XIC(ID0_ReceiveMSG1.DN) XIO(ID0_ReceiveMSG2.DN) MSG(ID0_ReceiveMSG2) ,XIC(ID0_ReceiveMSG2.DN) XIO(ID0_ReceiveMSG3.DN) MSG(ID0_ReceiveMSG3) ,[XIC(ID0_ReceiveMSG1.DN) XIC(ID0_ReceiveMSG2.DN) XIC(ID0_ReceiveMSG3.DN) CPS(RCP1_00.MISC.ParameterArray_RX_TX[0],RCP1_00.MISC.ParameterArray[0],RCP1_00.MISC.ParameterBytes) ,XIC(ID0_ReceiveMSG1.ER) OTU(ID0_ReceiveMSG1.ER) ,XIC(ID0_ReceiveMSG2.ER) OTU(ID0_ReceiveMSG2.ER) ,XIC(ID0_ReceiveMSG3.ER) OTU(ID0_ReceiveMSG3.ER) ] OTU(ID0_ReceiveMSG1.DN) OTU(ID0_ReceiveMSG2.DN) OTU(ID0_ReceiveMSG3.DN) OTU(RCP1_00.ReadParameter) ];
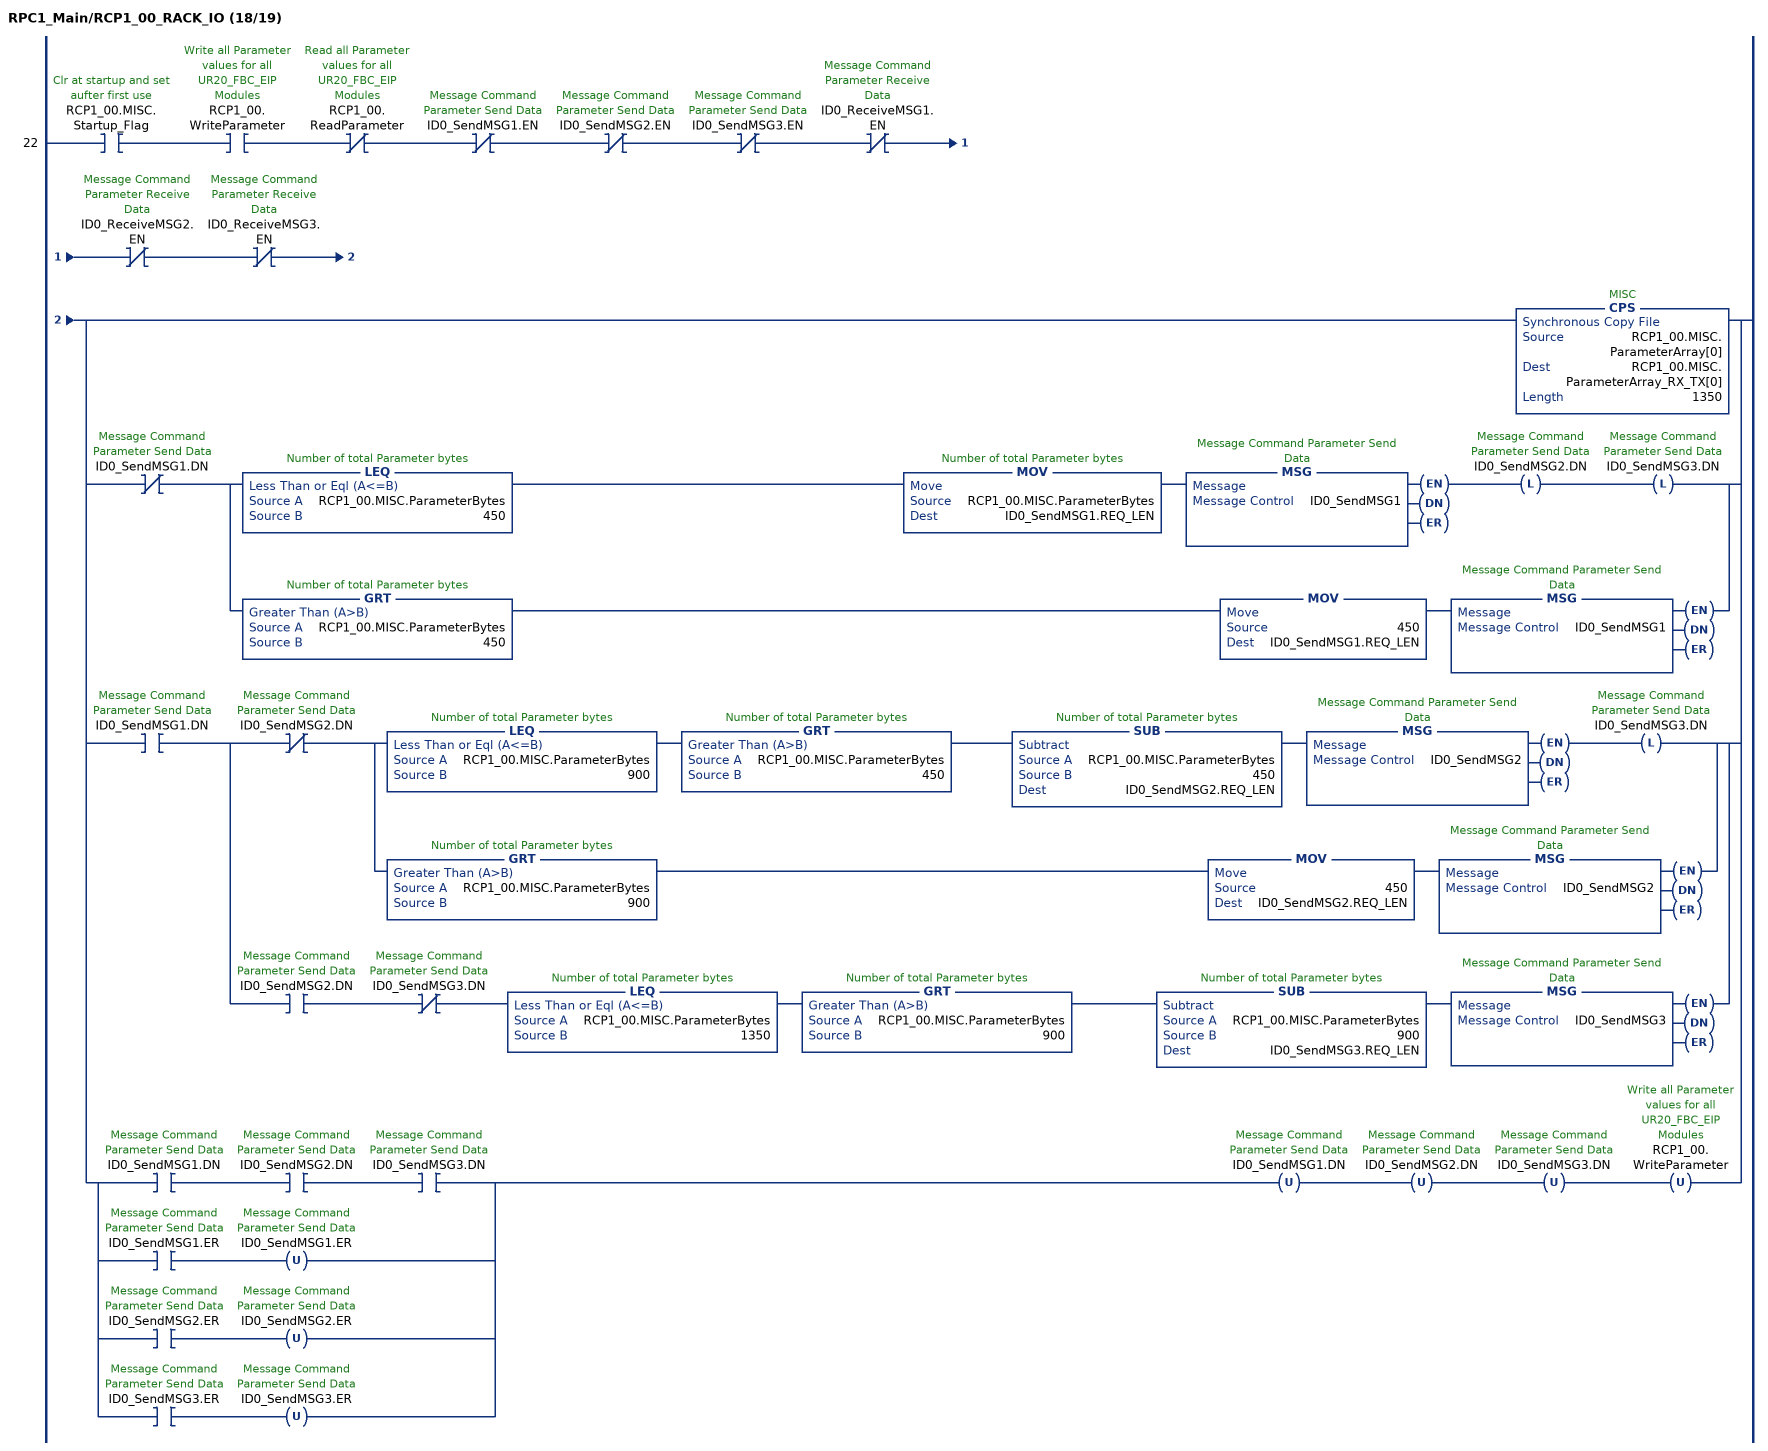
   22: XIC(RCP1_00.MISC.Startup_Flag)XIC(RCP1_00.WriteParameter)XIO(RCP1_00.ReadParameter)XIO(ID0_SendMSG1.EN)XIO(ID0_SendMSG2.EN)XIO(ID0_SendMSG3.EN)XIO(ID0_ReceiveMSG1.EN)XIO(ID0_ReceiveMSG2.EN)XIO(ID0_ReceiveMSG3.EN)[CPS(RCP1_00.MISC.ParameterArray[0],RCP1_00.MISC.ParameterArray_RX_TX[0],1350) ,[XIO(ID0_SendMSG1.DN) [LEQ(RCP1_00.MISC.ParameterBytes,450) MOV(RCP1_00.MISC.ParameterBytes,ID0_SendMSG1.REQ_LEN) MSG(ID0_SendMSG1) OTL(ID0_SendMSG2.DN) OTL(ID0_SendMSG3.DN) ,GRT(RCP1_00.MISC.ParameterBytes,450) MOV(450,ID0_SendMSG1.REQ_LEN) MSG(ID0_SendMSG1) ] ,XIC(ID0_SendMSG1.DN) [XIO(ID0_SendMSG2.DN) [LEQ(RCP1_00.MISC.ParameterBytes,900) GRT(RCP1_00.MISC.ParameterBytes,450) SUB(RCP1_00.MISC.ParameterBytes,450,ID0_SendMSG2.REQ_LEN) MSG(ID0_SendMSG2) OTL(ID0_SendMSG3.DN) ,GRT(RCP1_00.MISC.ParameterBytes,900) MOV(450,ID0_SendMSG2.REQ_LEN) MSG(ID0_SendMSG2) ] ,XIC(ID0_SendMSG2.DN) XIO(ID0_SendMSG3.DN) LEQ(RCP1_00.MISC.ParameterBytes,1350) GRT(RCP1_00.MISC.ParameterBytes,900) SUB(RCP1_00.MISC.ParameterBytes,900,ID0_SendMSG3.REQ_LEN) MSG(ID0_SendMSG3) ] ,[XIC(ID0_SendMSG1.DN) XIC(ID0_SendMSG2.DN) XIC(ID0_SendMSG3.DN) ,XIC(ID0_SendMSG1.ER) OTU(ID0_SendMSG1.ER) ,XIC(ID0_SendMSG2.ER) OTU(ID0_SendMSG2.ER) ,XIC(ID0_SendMSG3.ER) OTU(ID0_SendMSG3.ER) ] OTU(ID0_SendMSG1.DN) OTU(ID0_SendMSG2.DN) OTU(ID0_SendMSG3.DN) OTU(RCP1_00.WriteParameter) ] ];
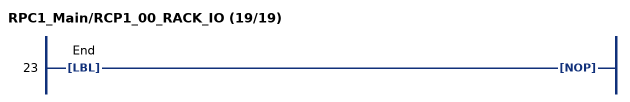
   23: LBL(End)NOP();
END_ROUTINE
END_PROGRAM
